Staubli VAL3: start.pgx

program start()
begin
  call Variables()
  call IO()
  call Deplacement()
end
